{attribute addProperty BoxType "EM7004-0000-0017"}
{attribute addProperty Id "DI_InputsAT %I*DI_Inputs_F7D3B19E1620ENC_Inputs_ChannelAT %I*ARRAY[0..3] OF ENC_Inputs_Channel_51DA946D192240PLS_InputsAT %I*PLS_Inputs_5BCA199F1620DO_OutputsAT %Q*DO_Outputs_6A0082531620AO_Outputs_ChannelAT %Q*ARRAY[0..3] OF AO_Outputs_Channel_F57FA4F96480ENC_Outputs_ChannelAT %Q*ARRAY[0..3] OF ENC_Outputs_Channel_5C86AA9D128160PLS_OutputsAT %Q*PLS_Outputs_D8F7BCB01620WcStateAT %I*WcState_98A4DF7520.250InfoDataAT %I*InfoData_BC63D37F80100"}
{attribute addProperty CRC "3573140132"}
{attribute addProperty SizeInBites "530"}
{attribute addProperty SizeInBytes "66.25"}
TYPE EM7004_7DC99940 :
STRUCT
	{attribute addProperty Name "DI_Inputs"}
	DI_Inputs : DI_Inputs_F7D3B19E;
	{attribute addProperty Name "ENC_Inputs_Channel"}
	ENC_Inputs_Channel : ARRAY[0..3] OF ENC_Inputs_Channel_51DA946D;
	{attribute addProperty Name "PLS_Inputs"}
	PLS_Inputs : PLS_Inputs_5BCA199F;
	{attribute addProperty Name "DO_Outputs"}
	DO_Outputs : DO_Outputs_6A008253;
	{attribute addProperty Name "AO_Outputs_Channel"}
	AO_Outputs_Channel : ARRAY[0..3] OF AO_Outputs_Channel_F57FA4F9;
	{attribute addProperty Name "ENC_Outputs_Channel"}
	ENC_Outputs_Channel : ARRAY[0..3] OF ENC_Outputs_Channel_5C86AA9D;
	{attribute addProperty Name "PLS_Outputs"}
	PLS_Outputs : PLS_Outputs_D8F7BCB0;
	{attribute addProperty Name "WcState"}
	WcState : WcState_98A4DF75;
	{attribute addProperty Name "InfoData"}
	InfoData : InfoData_BC63D37F;
END_STRUCT
END_TYPE

(* stored: Version 1.2.0.0, ProductVersion 3.1.4024.9
   DUT EM7004_7DC99940: Id {7c46a517-2101-4d19-9315-775f37aa5a2b} *)
